{attribute addProperty BoxType "EL5032-0000-0021"}
{attribute addProperty Id "WarningBIT10.1251ErrorBIT10.1252ReadyBIT10.1253DiagBIT10.12513TxPDO_StateBIT10.12514Input_cycle_counter_BIT_0BIT10.12515Input_cycle_counter_BIT_1BIT10.12515"}
{attribute addProperty CRC "4110715007"}
{attribute addProperty SizeInBites "16"}
{attribute addProperty SizeInBytes "2"}
TYPE Status_F504887F :
STRUCT
	{attribute addProperty Name "Warning"}
	Warning : BIT;
	{attribute addProperty Name "Error"}
	Error : BIT;
	{attribute addProperty Name "Ready"}
	Ready : BIT;
	{attribute 'hide'}
	reserve_1_BIT_0 : BIT;
	{attribute 'hide'}
	reserve_1_BIT_1 : BIT;
	{attribute 'hide'}
	reserve_1_BIT_2 : BIT;
	{attribute 'hide'}
	reserve_1_BIT_3 : BIT;
	{attribute 'hide'}
	reserve_1_BIT_4 : BIT;
	{attribute 'hide'}
	reserve_2_BIT_0 : BIT;
	{attribute 'hide'}
	reserve_2_BIT_1 : BIT;
	{attribute 'hide'}
	reserve_2_BIT_2 : BIT;
	{attribute 'hide'}
	reserve_2_BIT_3 : BIT;
	{attribute addProperty Name "Diag"}
	Diag : BIT;
	{attribute addProperty Name "TxPDO_State"}
	TxPDO_State : BIT;
	{attribute addProperty Name "Input_cycle_counter"}
	Input_cycle_counter_BIT_0 : BIT;
	{attribute addProperty Name "Input_cycle_counter"}
	Input_cycle_counter_BIT_1 : BIT;
END_STRUCT
END_TYPE

(* stored: Version 1.2.0.0, ProductVersion 3.1.4024.9
   DUT Status_F504887F: Id {c024c737-30e0-4174-b070-b1d548e8defb} *)
